//==================================================================================================
//							Beckhoff Automation Poland
//									18.04.2018
//	Struktura zawierajaca I/O odpowiedniego bloku
//  v1.0	|| TC v 3.1.4022.16		|| - pierwsza wersja
//==================================================================================================
TYPE ST_MCStopIO:
STRUCT
	bExecute						: BOOL;								// Rising edge executes cmd
	lrDeceleration					: LREAL; 
	lrJerk							: LREAL;
	stOptions						: Tc2_MC2.ST_MoveOptions;
	bDone							: BOOL;
	bBusy							: BOOL;
	bActive							: BOOL;
	bCommandAborted					: BOOL;
	bError							: BOOL;
	udiErrorID						: UDINT;
END_STRUCT
END_TYPE

(* stored: Version 1.1.0.1, ProductVersion 3.1.4022.12
   DUT ST_MCStopIO: Id {1ae26df7-6fdc-4f88-bb98-8df3c4bb7f5f} *)
